PROGRAM P_CP1_Check
VAR
END_VAR

END_PROGRAM

(* stored: Version 1.1.0.1, ProductVersion 3.1.4024.15
   POU P_CP1_Check: Id {6176801c-fa9a-48a4-9f5e-14dd91aa3a80}, SpecialFunc None *)
